(* IEC 61131-3 sources: WarwickBoringPLC/Safety, 7 files *)

(* ---- systemGVL.gvl ---- *)
{attribute 'qualified_only'}
VAR_GLOBAL
    // Whole system state
    systemState:  SYSTEM_STATE := SYSTEM_STATE.NULL;
    finishedInitialising: BOOL := FALSE; //high when PLC ready to run
    resetSignal:  BOOL := FALSE; //high when PLC should reset
    finishedResetting:     BOOL := FALSE; //high when PLC has reset
    startSignal:  BOOL := FALSE; //high when PLC should start
    finishedStarting:   BOOL := FALSE; //high when PLC has started
    suspendSignal: BOOL := FALSE; //high when PLC should suspend
    finishedSuspending: BOOL := FALSE; //high when PLC has suspended
    unsuspendSignal : BOOL := FALSE; //high when PLC should unsuspend
    finishedUnsuspending: BOOL := FALSE; //high when PLC has unsuspended
    stopSignal:   BOOL := FALSE; //high when PLC should stop
    finishingStopping:   BOOL := FALSE; //high when PLC has stopped
    abortSignal:  BOOL := FALSE; //high when PLC should abort
    finishedAborting:   BOOL := FALSE; //high when PLC has aborted
    clearSignal: BOOL := FALSE; //high when PLC should clear
    resetTrigger: R_TRIG;
    startTrigger: R_TRIG;
    suspendTrigger: R_TRIG;
    unsuspendTrigger: R_TRIG;
    stoppingTrigger: R_TRIG;
    abortTrigger: R_TRIG;
    clearTrigger: R_TRIG;
    stateError:  BOOL := FALSE; //high when PLC was in an invalid state
END_VAR

(* ---- stateToText.st ---- *)
FUNCTION_BLOCK stateToString
VAR_INPUT
    state : SYSTEM_STATE;
END_VAR
VAR_OUTPUT
    stateString : STRING;
END_VAR

CASE state OF
    SYSTEM_STATE.NULL:
        stateString := 'NULL';
    SYSTEM_STATE.INITIALISING:
        stateString := 'INITIALISING';
    SYSTEM_STATE.STOPPED:
        stateString := 'STOPPED';
    SYSTEM_STATE.RESETTING:
        stateString := 'RESETTING';
    SYSTEM_STATE.IDLE:
        stateString := 'IDLE';
    SYSTEM_STATE.STARTING:
        stateString := 'STARTING';
    SYSTEM_STATE.RUNNING:
        stateString := 'RUNNING';
    SYSTEM_STATE.SUSPENDING:
        stateString := 'SUSPENDING';
    SYSTEM_STATE.SUSPENDED:
        stateString := 'SUSPENDED';
    SYSTEM_STATE.UNSUSPENDING:
        stateString := 'UNSUSPENDING';
    SYSTEM_STATE.STOPPING:
        stateString := 'STOPPING';
    SYSTEM_STATE.ABORTING:
        stateString := 'ABORTING';
    SYSTEM_STATE.ABORTED:
        stateString := 'ABORTED';
    SYSTEM_STATE.CLEARING:
        stateString := 'CLEARING';
    ELSE
        stateString := 'ERROR';
END_CASE

(* ---- TBMHeartbeat.st ---- *)
FUNCTION_BLOCK
    VAR
        beatTOF : TOF;
    END_VAR
    //rising edge rests timer
    //mGVL.tbmStatusIn

    beatTOF(IN := mGVL.tbmStatusIn, PT:= T#1s, Q => mainGVL.tbmPIHeartBeat); //low after 1s if no heartbeat

END_FUNCTION_BLOCK

(* ---- isUnsafe.st ---- *)
PROGRAM safety

END_PROGRAM

FUNCTION isUnsafe : BOOL
    VAR_INPUT
        sensorValue: REAL; (* sensor input value *)
        sensorMax: REAL; (* max safe value the sensor can take *)
        sensorMin: REAL; (* min safe value the sensor can take *)
    END_VAR
    VAR_OUTPUT
        unSafe: BOOL; (* is the value safe *)
    END_VAR

    IF sensorValue > sensorMax OR sensorValue < sensorMin THEN
        unSafe := TRUE;
    ELSE
        unSafe := FALSE;
    END_IF;
END_FUNCTION

(* ---- safteyProg.st ---- *)
PROGRAM SafetyProg
VAR
	isHPSA_unsafe : BOOL; // True if Hydraullic Pressure is too high
	isEStopPressed : BOOL; // True if an ESTOP is pressed

END_VAR

// Safety runs as a seperate task checking for interlocks, seperate to the main task to prevent stalls.

// Hydraulic Pressure Sensor A
isUnsafe(sensorMin := - 26, sensorMax := 100, sensorValue := mgvl.hydraulicPressureSensorA, unSafe => isHPSA_unsafe);

// Control Cabinet E STOP, Visualisation Estop
isEStopPressed := (NOT mgvl.eStopCC) OR visuGVL.visuEstop;

mainGVL.isIssue := isHPSA_unsafe OR isESTOPPressed;

// Interlock Check
IF mainGVL.isIssue THEN
	mainGVL.isSystemInterlocked := TRUE;
END_IF

mainGVL.isResettable := (NOT mainGVL.isIssue) AND (mainGVL.isSystemInterlocked);

// If clearable, and then reset button pressed
IF mainGVL.isResettable AND (visuGVL.resetButton) THEN
	// Then reset estop
	mainGVL.isSystemInterlocked := FALSE;

END_IF

(* ---- stateVars.st ---- *)
//declare vars
VAR
    resetTP : TP;
    resetTON : TON;
    stoppingTP : TP;
    stoppingTON : TON;
    suspendingTP : TP;
    suspendingTON : TON;
    unsuspendingTP : TP;
    unsuspendingTON : TON;
END_VAR

//each timer 2s

//init vars
resetTP (IN:= systemGVL.resetTrigger.Q, PT := T#3s);
resetTON (IN:= resetTP.Q, PT := T#2s);
stoppingTP (IN:= systemGVL.stoppingTrigger.Q, PT := T#3s);
stoppingTON (IN:= stoppingTP.Q, PT := T#2s);
suspendingTP (IN:= systemGVL.suspendingTrigger.Q, PT := T#3s);
suspendingTON (IN:= suspendingTP.Q, PT := T#2s);
unsuspendingTP (IN:= systemGVL.unsuspendingTrigger.Q, PT := T#3s);
unsuspendingTON (IN:= unsuspendingTP.Q, PT := T#2s);
startingTP (IN:= systemGVL.startingTrigger.Q, PT := T#3s);
startingTON (IN:= startingTP.Q, PT := T#2s);

//logic
IF systemGVL.SYSTEM_STATE >= 0 THEN

    systemGVL.finishedInitialising := TRUE;

    systemGVL.finishedResetting := resetTON.Q;

    //systemGVL.finishedStarting
    //read pressures, ensure they are in expected range
    //1 if pressure good, 0 if not

    //systemGVL.finishedSuspending
    //read valve positions, should be closed
    //1 if closed, 0 if not

    systemGVL.finishedUnsuspending := TRUE;
    //as no tunnel lining, nothing happens in unsuspending state - skip to next state
    //read valves, should be opening again
    //1 if open, 0 if not

    //systemGVL.finishedStopping
    //read ME, TL power states, should be off
    //read hydraulics, keep on
    //read pressures, ensure depressurised
    //1 if so, 0 if not

    //systemGVL.finishedAborting
    //ME power off
    //TL power off
    //hydraulics power on, relief valve open, depressurised
    //1 if so, 0 if not

END_IF

(* ---- SystemStateMachine.st ---- *)
systemGVL.resetTrigger (CLK := systemGVL.resetSignal); //reset trigger
systemGVL.startTrigger (CLK := systemGVL.startSignal); //start trigger
systemGVL.suspendTrigger (CLK := systemGVL.suspendSignal); //suspend trigger
systemGVL.unsuspendTrigger (CLK := systemGVL.unsuspendSignal); //unsuspend trigger
systemGVL.clearTrigger (CLK := systemGVL.clearSignal); //clear trigger
systemGVL.abortTrigger (CLK := systemGVL.abortSignal); //abort trigger
systemGVL.stopTrigger (CLK := systemGVL.stopSignal); //stop trigger

CASE systemGVL.systemState OF
    SYSTEM_STATE.NULL:
        systemGVL.systemState := SYSTEM_STATE.INIT; //move to initialise
    SYSTEM_STATE.INITIALISING:
        IF systemGVL.finishedInitialising THEN
            systemGVL.systemState := SYSTEM_STATE.STOPPED; //move to stopped
        END_IF
    SYSTEM_STATE.STOPPED:
        IF systemGVL.resetTrigger.Q THEN
            systemGVL.systemState := SYSTEM_STATE.RESETTING; //move to resetting
        END_IF
    SYSTEM_STATE.RESETTING:
        IF systemGVL.finishedResetting THEN
            systemGVL.systemState := SYSTEM_STATE.IDLE; //move to isle
        END_IF
    SYSTEM_STATE.IDLE:
        IF systemGVL.startTrigger.Q THEN
            systemGVL.systemState := SYSTEM_STATE.STARTING; //move to starting
        END_IF
    SYSTEM_STATE.STARTING:
        IF systemGVL.finishedStarting THEN
            systemGVL.systemState := SYSTEM_STATE.RUNNING; //move to running
        END_IF
    SYSTEM_STATE.RUNNING:
        IF systemGVL.suspendTrigger.Q THEN
            systemGVL.systemState := SYSTEM_STATE.SUSPENDING; //move to suspending
        END_IF
    SYSTEM_STATE.SUSPENDING:
        IF systemGVL.finishedSuspending THEN
            systemGVL.systemState := SYSTEM_STATE.SUSPENDED; //move to suspended
        END_IF
    SYSTEM_STATE.SUSPENDED:
        IF systemGVL.unsuspendTrigger.Q THEN
            systemGVL.systemState := SYSTEM_STATE.UNSUSPENDING; //move to unsuspending
        END_IF
    SYSTEM_STATE.UNSUSPENDING:
        IF systemGVL.finishedUnsuspending THEN
            systemGVL.systemState := SYSTEM_STATE.RUNNING; //move to running
        END_IF
    SYSTEM_STATE.STOPPING:
        IF systemGVL.finishingStopping THEN
            systemGVL.systemState := SYSTEM_STATE.STOPPED; //move to stopped
        END_IF
    SYSTEM_STATE.ABORTING:
        IF systemGVL.finishedAborting THEN
            systemGVL.systemState := SYSTEM_STATE.ABORTED; //move to stopped
        END_IF
    SYSTEM_STATE.ABORTED:
        IF systemGVL.clearTrigger.Q THEN
            systemGVL.systemState := SYSTEM_STATE.CLEARING; //move to clearing
        END_IF
    SYSTEM_STATE.CLEARING:
        IF systemGVL.isCleared THEN
            systemGVL.systemState := SYSTEM_STATE.STOPPED; //move to stopped
        END_IF
    ELSE:
        systemGVL.systemState := SYSTEM_STATE.ABORTING; //error has occured
        systemGVL.stateError := TRUE;
END_CASE

IF systemGVL.abortTrigger.Q THEN
    systemGVL.systemState := SYSTEM_STATE.ABORTING; //move to aborting
ELSEIF systemGVL.stopTrigger.Q THEN
    systemGVL.systemState := SYSTEM_STATE.STOPPING; //move to stopping
END_IF
